Yaskawa INFORM job: X2_57-69(2)(90,180).JBI

/JOB
//NAME X2_57-69(2)(90,180)
//POS
///NPOS 364,364,364,19,0,0
///TOOL 0
///POSTYPE PULSE
///PULSE
C00000=-2000,-108350,-112464,0,80055,0
C00001=117728,-108350,-112464,34609,80055,28580
C00002=124329,53851,34766,36826,59228,24303
C00003=124742,48200,29458,35015,59253,25605
C00004=132091,87021,68515,19398,44781,35491
C00005=131964,91219,74916,20112,43130,35046
C00006=131964,92220,77875,20603,41902,34745
C00007=131925,92203,77341,20509,42211,34802
C00008=131397,96741,83157,21411,41178,34254
C00009=131925,92203,77341,20509,42211,34802
C00010=132378,78684,56627,18262,47592,36223
C00011=132682,70057,46287,17529,49367,36706
C00012=119143,48210,55676,30149,44593,-20608
C00013=119357,47156,53956,26116,42767,-17551
C00014=120340,57080,66927,26977,39866,-17985
C00015=120719,61633,72965,27509,38514,-18256
C00016=120718,63903,77470,28475,37088,-18806
C00017=120500,60851,73214,27972,38091,-18544
C00018=120914,65321,78494,28289,37111,-18678
C00019=120500,60851,73214,27972,38091,-18544
C00020=119122,46332,54187,26526,42331,-17820
C00021=118999,38480,45168,29507,46176,-20252
C00022=119368,-115903,-71302,26914,50601,-18610
C00023=64607,-7982,-59747,-18064,104585,18556
C00024=122352,27346,-5631,2134,105537,41861
C00025=121432,26579,-2459,2110,103216,41509
C00026=121064,26360,-1109,2102,102282,41368
C00027=120094,26356,-1113,2104,102307,41040
C00028=120094,26183,380,2095,101300,41022
C00029=120094,26356,-1113,2104,102307,41040
C00030=121064,26360,-1109,2102,102282,41368
C00031=121064,26166,399,2092,101255,41350
C00032=120526,26160,392,2094,101269,41168
C00033=121064,26166,399,2092,101255,41350
C00034=121064,26360,-1109,2102,102282,41368
C00035=121432,26579,-2459,2110,103216,41509
C00036=122352,27346,-5631,2134,105537,41861
C00037=122404,27316,-5660,2134,105538,41879
C00038=121484,26548,-2490,2110,103217,41527
C00039=121116,26328,-1140,2102,102284,41386
C00040=119990,26323,-1145,2104,102313,41004
C00041=119990,26151,349,2095,101305,40987
C00042=119990,26323,-1145,2104,102313,41004
C00043=121116,26328,-1140,2102,102284,41386
C00044=121116,26236,467,2092,101248,41368
C00045=120578,26229,460,2094,101262,41186
C00046=121116,26236,467,2092,101248,41368
C00047=121116,26328,-1140,2102,102284,41386
C00048=121484,26548,-2490,2110,103217,41527
C00049=122404,27316,-5660,2134,105538,41879
C00050=64607,-7982,-59747,-18064,104585,18556
C00051=43259,-142284,-94849,68481,67043,45987
C00052=75789,-57542,-35879,68380,64193,60275
C00053=79378,-55423,-31936,68889,61283,60160
C00054=80801,-54484,-30299,69115,60133,60112
C00055=80803,-53463,-27973,69597,59790,59668
C00056=80780,-53792,-28606,69479,59888,59772
C00057=82380,-55228,-29381,69587,58724,59873
C00058=80801,-53699,-28530,69478,59874,59776
C00059=81788,-51404,-27272,69234,59369,60118
C00060=80801,-53699,-28530,69478,59874,59776
C00061=79378,-54655,-30185,69233,61022,59829
C00062=75790,-56818,-34168,68680,63927,59955
C00063=84853,-69188,-42023,59966,34850,64425
C00064=87616,-64026,-36454,59770,32751,64733
C00065=88672,-61932,-34175,59731,31934,64834
C00066=88674,-60834,-31833,60968,31481,64183
C00067=88651,-60985,-32132,60826,31549,64256
C00068=90372,-59623,-31443,59618,30637,65026
C00069=88651,-60985,-32132,60826,31549,64256
C00070=87595,-63088,-34428,60823,32369,64172
C00071=84831,-68269,-40036,60922,34477,63902
C00072=34135,-92769,-74242,67244,95299,48930
C00073=35401,-42276,-48954,68810,98599,53574
C00074=65945,-1100,7259,69270,87048,42040
C00075=68239,35,11214,69501,84806,41537
C00076=69159,585,12885,69624,83908,41331
C00077=69161,1574,15470,69708,83504,40864
C00078=69221,1430,14991,69696,83546,40967
C00079=70472,2033,15498,69808,82706,41122
C00080=69221,1430,14991,69696,83546,40967
C00081=68301,843,13280,69560,84443,41175
C00082=66008,-382,9232,69294,86686,41685
C00083=65045,17742,23285,68512,88220,38243
C00084=67089,19246,27753,68708,86083,37667
C00085=67908,20664,31476,68858,84932,37105
C00086=67909,21636,33893,68917,84551,36681
C00087=67870,21286,33093,68893,84697,36810
C00088=69603,21321,33122,69077,83544,37032
C00089=67870,21286,33093,68893,84697,36810
C00090=67052,20507,31108,68763,85558,37056
C00091=65008,18839,26451,68515,87704,37647
C00092=35401,-42276,-48954,68810,98599,53574
C00093=34135,-92769,-74242,67244,95299,48930
C00094=40047,-44089,-55446,21687,109798,-38511
C00095=62225,-62197,-88507,27498,109393,-46828
C00096=110162,-85165,-68253,22495,93568,-66447
C00097=113189,-87083,-65902,22697,90484,-65921
C00098=114452,-87710,-64890,22792,89260,-65692
C00099=114517,-85766,-62478,22795,88793,-65757
C00100=114452,-87710,-64890,22792,89260,-65692
C00101=114560,-85938,-62764,22799,88863,-65728
C00102=116855,-86136,-62847,22980,88180,-65021
C00103=114560,-85938,-62764,22799,88863,-65728
C00104=116037,-86901,-63721,22918,88541,-65250
C00105=115908,-89550,-64185,22909,87583,-65481
C00106=116037,-86901,-63721,22918,88541,-65250
C00107=114760,-86329,-64757,22823,89756,-65485
C00108=111694,-84556,-67168,22619,92819,-66026
C00109=100686,-82782,-64085,34767,78413,-50947
C00110=101124,-84756,-62575,46086,58567,-32836
C00111=105363,-79670,-59021,44782,56711,-31479
C00112=106963,-77579,-57544,44243,56028,-30951
C00113=107094,-75757,-55111,44466,55555,-31127
C00114=106963,-77579,-57544,44243,56028,-30951
C00115=107061,-76131,-55605,44423,55653,-31093
C00116=109164,-76621,-55827,43839,54522,-30514
C00117=107061,-76131,-55605,44423,55653,-31093
C00118=152521,-89404,-55591,-46164,31260,15215
C00119=151593,-87290,-55392,-44387,31486,14209
C00120=152521,-89404,-55591,-46164,31260,15215
C00121=153310,-92374,-57074,-47433,31236,15946
C00122=155515,-99823,-60624,-50849,31303,17939
C00123=144863,-106519,-66042,-48559,45403,33907
C00124=128223,-91539,-64179,-39651,61078,44936
C00125=123361,-87629,-60570,-38638,58731,43541
C00126=121491,-85978,-59075,-38202,57849,42987
C00127=121484,-83973,-56613,-38386,57460,43144
C00128=121491,-85978,-59075,-38202,57849,42987
C00129=121461,-84428,-57196,-38332,57549,43096
C00130=119429,-85653,-57392,-38005,56255,42626
C00131=121461,-84428,-57196,-38332,57549,43096
C00132=119967,-84308,-57809,-37774,57245,42484
C00133=118856,-82106,-57411,-37133,57477,41844
C00134=119967,-84308,-57809,-37774,57245,42484
C00135=121794,-85994,-59329,-38223,58099,43033
C00136=126552,-90004,-63001,-39273,60372,44418
C00137=126573,-96663,-78450,-37396,65213,42514
C00138=131304,-91681,-76533,-26004,78425,57156
C00139=124056,-87914,-75121,-11214,89260,70181
C00140=122142,-89367,-72002,-11215,86376,69779
C00141=121349,-89811,-70686,-11221,85247,69607
C00142=121343,-87912,-68316,-11227,84773,69647
C00143=121349,-89811,-70686,-11221,85247,69607
C00144=121327,-88368,-69271,-11223,85117,69610
C00145=121333,-89533,-69503,-11227,84670,69652
C00146=121327,-88658,-70019,-11219,85423,69583
C00147=119585,-89190,-70235,-11210,85043,69016
C00148=122145,-87062,-69869,-11216,86251,69790
C00149=120261,-90277,-71864,-11211,85572,69201
C00150=122240,-88980,-75059,-11209,88432,69628
C00151=122263,-92131,-88871,-11297,95190,69025
C00152=118027,-102145,-112609,12133,81631,15728
C00153=114779,-111065,-98137,30741,51344,-26323
C00154=118307,-102289,-93656,28063,51644,-24513
C00155=119601,-98864,-91828,27075,51783,-23857
C00156=119613,-97097,-89588,27235,51358,-23975
C00157=119601,-98864,-91828,27075,51783,-23857
C00158=110485,-79839,-84525,36111,67748,-27732
C00159=112543,-80296,-84732,35339,66815,-27160
C00160=110485,-79839,-84525,36111,67748,-27732
C00161=133496,-108715,-92181,7385,37609,-14213
C00162=133101,-105069,-91479,7525,39076,-14289
C00163=133496,-108715,-92181,7385,37609,-14213
C00164=132876,-112861,-94058,8163,36703,-14650
C00165=131137,-123655,-98655,10535,34221,-15975
C00166=123443,-118355,-110381,19336,67280,-34215
C00167=114391,-92529,-101967,29874,101827,-55519
C00168=118393,-95739,-100418,29397,98177,-54940
C00169=120031,-96781,-99698,29226,96757,-54678
C00170=120038,-95275,-97552,29185,96274,-54799
C00171=120031,-96781,-99698,29226,96757,-54678
C00172=120084,-95528,-97941,29191,96355,-54761
C00173=122387,-95485,-97926,29054,95580,-54078
C00174=120084,-95528,-97941,29191,96355,-54761
C00175=120976,-97030,-99100,29136,95998,-54511
C00176=120991,-101427,-100201,29036,94603,-54858
C00177=120976,-97030,-99100,29136,95998,-54511
C00178=119331,-96066,-99851,29302,97402,-54781
C00179=115306,-93056,-101481,29762,101015,-55383
C00180=119500,-95286,-111088,6725,93490,-23573
C00181=126773,-109990,-105967,-32242,60764,29595
C00182=122699,-100871,-93398,-31267,56629,29081
C00183=121186,-97859,-91654,-30361,56488,28429
C00184=121181,-96122,-89420,-30519,56067,28559
C00185=121186,-97859,-91654,-30361,56488,28429
C00186=121151,-96393,-89780,-30476,56128,28526
C00187=118823,-96364,-89767,-29286,55307,27705
C00188=121151,-96393,-89780,-30476,56128,28526
C00189=120304,-96962,-90655,-29967,56039,28163
C00190=120309,-93163,-89734,-29527,57250,27795
C00191=120304,-96962,-90655,-29967,56039,28163
C00192=121790,-99973,-92408,-30869,56167,28809
C00193=125792,-107589,-96692,-33228,56592,30543
C00194=131625,-94984,-104332,-26399,91581,50246
C00195=126745,-145288,-119778,-15495,97214,71135
C00196=123697,-150191,-117695,-15760,92961,70600
C00197=122386,-151760,-116729,-15896,91357,70347
C00198=122362,-148095,-114205,-15905,91670,70298
C00199=122386,-151760,-116729,-15896,91357,70347
C00200=152021,-159898,-112636,-26025,88694,79156
C00201=148454,-161901,-113048,-26644,86894,78253
C00202=152021,-159898,-112636,-26025,88694,79156
C00203=97626,-122802,-108845,-7114,105595,63457
C00204=96843,-127398,-109672,-7190,103687,63292
C00205=97626,-122802,-108845,-7114,105595,63457
C00206=98540,-120520,-109456,-7005,107212,63690
C00207=100688,-114056,-110651,-6782,111424,64223
C00208=141928,-132033,-122827,-28072,87297,56565
C00209=127745,-107087,-104050,-36954,70100,33758
C00210=123019,-101123,-100201,-35200,68701,32195
C00211=121229,-98695,-98613,-34495,68204,31593
C00212=121224,-97088,-96437,-34605,67775,31733
C00213=121229,-98695,-98613,-34495,68204,31593
C00214=121227,-97196,-96702,-34583,67865,31704
C00215=118899,-97170,-96690,-33712,66948,31006
C00216=121227,-97196,-96702,-34583,67865,31704
C00217=120189,-96862,-97597,-34041,68055,31198
C00218=120197,-92600,-96484,-33733,69318,30794
C00219=120189,-96862,-97597,-34041,68055,31198
C00220=121940,-99293,-99200,-34743,68533,31788
C00221=126568,-105279,-103092,-36497,69877,33324
C00222=126928,-101255,-99744,-25325,80548,44815
C00223=122663,-98736,-96036,-24420,78380,43689
C00224=120996,-97606,-94499,-24052,77561,43237
C00225=120993,-95941,-92294,-24092,77100,43331
C00226=120996,-97606,-94499,-24052,77561,43237
C00227=121020,-96262,-92743,-24089,77210,43319
C00228=118702,-96225,-92727,-23520,76555,42587
C00229=121020,-96262,-92743,-24089,77210,43319
C00230=122674,-97386,-94282,-24452,78030,43766
C00231=126903,-99897,-97999,-25343,80198,44881
C00232=120621,-96600,-101484,-24088,62946,45857
C00233=120621,-96804,-99274,-24394,61605,46162
C00234=121065,-96725,-98290,-24739,61217,46434
C00235=120808,-96049,-104031,-23738,79088,41099
C00236=120748,-96229,-90224,-24572,71199,42719
C00237=112992,-105726,-101839,-14067,93209,37194
C00238=115215,-122388,-108196,-15088,94657,37910
C00239=120621,-96757,-99844,-19967,111704,37232
C00240=139470,-90927,-100236,-32127,92639,54211
C00241=120586,-139946,-100537,-59993,22470,77721
C00242=120585,-131753,-89573,-65663,21254,80445
C00243=120585,-129979,-87167,-67023,21013,81095
C00244=120562,-131266,-88538,-66553,21075,80878
C00245=122227,-132208,-89206,-62791,23886,78792
C00246=121243,-147626,-110329,-33756,48909,60234
C00247=120920,-140051,-100583,-34677,47022,60829
C00248=124359,-147547,-111068,-11567,101442,53176
C00249=120588,-147693,-110556,-9391,106075,51659
C00250=120588,-150839,-114378,-9432,106801,51602
C00251=120668,-127498,-127599,8027,92338,11843
C00252=106540,-131828,-115388,26739,62994,-22536
C00253=120606,-112501,-85686,37507,17849,-56930
C00254=120605,-109780,-80480,41231,16435,-58666
C00255=120605,-108994,-78986,42415,16045,-59215
C00256=120315,-109307,-78838,43536,15999,-59746
C00257=120588,-122985,-110649,24761,70026,-42850
C00258=120328,-120662,-104365,25254,67672,-43482
C00259=120364,-122737,-110073,20558,99126,-39146
C00260=120608,-123337,-111674,20610,99768,-38950
C00261=120609,-124066,-114983,20744,101328,-38677
C00262=120610,-124421,-123392,21260,106003,-37833
C00263=120649,-125888,-127056,5137,96316,-15534
C00264=120651,-130620,-101533,-26318,65901,27317
C00265=132080,-98652,-65915,-40871,60604,46715
C00266=126739,-94814,-62411,-39928,58019,45199
C00267=125167,-93744,-61263,-39656,57186,44775
C00268=114973,-73674,-63266,-21215,75827,54043
C00269=129996,-102072,-68542,-24583,69504,61007
C00270=129963,-88454,-64083,-24262,79764,67113
C00271=119249,-73873,-63371,-13635,90655,67540
C00272=119873,-76495,-66852,-13633,91534,67660
C00273=119888,-78331,-76038,-13747,96118,67156
C00274=119081,-108028,-88031,16388,61795,15984
C00275=117234,-100128,-64028,47858,30144,-31364
C00276=117223,-96877,-58390,50267,28944,-32603
C00277=120408,-90078,-55153,45893,28312,-30090
C00278=121323,-87057,-53987,43493,28946,-29243
C00279=115884,-56336,-58001,25875,73139,-43981
C00280=110450,-120996,-68796,34057,51702,-52465
C00281=115886,-81683,-60397,23196,86120,-63160
C00282=116435,-73198,-57641,22557,92556,-65246
C00283=113722,-71149,-59788,22419,95499,-65689
C00284=113460,-61701,-78205,24579,95746,-61766
C00285=45876,-101964,-103313,26325,110018,-55581
C00286=15431,-40197,-19183,56345,102197,5038
C00287=34862,-44642,-10243,68104,90731,26909
C00288=38272,-42530,-5806,68888,87904,26638
C00289=46229,766,28384,61909,108262,28635
C00290=46231,618,28261,61910,108260,28636
C00291=41809,-20527,11988,64520,102557,33043
C00292=37345,-41369,-1566,65704,98540,31804
C00293=38123,-41321,-1546,64762,100173,32421
C00294=38612,-39929,-4176,63239,100836,34262
C00295=36669,-38826,-14631,64435,105300,36937
C00296=35614,-75221,-31334,66701,43579,46020
C00297=-4350,-87290,-51239,65137,72622,41765
C00298=64440,-113176,-91621,27014,43904,67647
C00299=122842,55452,53671,34630,66319,-4477
C00300=122836,62423,70424,36514,60793,-6445
C00301=123914,74645,87958,37956,56708,-7549
C00302=125197,76616,91296,38180,55337,-7504
C00303=125636,70432,83250,33590,52050,-4701
C00304=125796,66906,78975,31139,50064,-1893
C00305=125404,66054,77985,29591,48689,-234
C00306=125098,65276,77131,27878,47332,1494
C00307=124827,64021,75593,26067,46325,3194
C00308=126696,59695,70609,19763,43762,8616
C00309=131143,56273,67245,5204,39677,20871
C00310=133431,54832,66811,-3343,37312,26727
C00311=136536,53744,67301,-15167,35496,34368
C00312=138731,52021,65734,-21083,35846,38135
C00313=139736,44763,55186,-20533,38686,37917
C00314=132675,46810,50748,6411,52596,1677
C00315=131127,80601,47453,25263,64319,31877
C00316=132807,97166,57058,12495,61470,40417
C00317=132437,103413,60649,12594,62499,40395
C00318=132694,105523,62562,12460,62371,40474
C00319=135614,121161,83227,11303,57371,41050
C00320=136368,126562,90481,11059,55609,41167
C00321=135950,123674,72731,10332,64945,41919
C00322=131127,80601,47453,25263,64319,31877
C00323=64440,-113176,-91621,27014,43904,67647
C00324=-4350,-87290,-51239,65137,72622,41765
C00325=52724,-99155,-43299,70564,49554,58260
C00326=58609,-95164,-38578,71970,45609,58601
C00327=62335,-94288,-36780,73026,43083,58718
C00328=62099,-93953,-36639,72913,43256,58740
C00329=60961,-88486,-31404,79687,39616,52248
C00330=56515,-82230,-27602,80423,44365,48776
C00331=50142,-68435,-18604,81559,53334,41178
C00332=51696,-72558,-17243,91450,48356,32919
C00333=47167,-82165,-29359,87907,51434,34351
C00334=62742,-127620,-60643,64448,25144,51124
C00335=120681,-113766,-68295,5608,40697,75829
C00336=102629,-70164,-59862,1874,75871,45222
C00337=101346,-35641,-42715,497,87745,38363
C00338=108372,-47074,-47716,-765,88535,35936
C00339=106813,-45162,-42766,-663,86458,35421
C00340=106148,-44305,-40721,-618,85635,35200
C00341=108217,-21947,-25956,-755,88052,35887
C00342=108724,-23055,-28269,-789,88913,36052
C00343=110078,-24539,-33116,-879,91147,36494
C00344=108372,-47074,-47716,-765,88535,35936
C00345=106813,-45162,-42766,-663,86458,35421
C00346=106197,-44302,-40640,-622,85587,35216
C00347=108187,-22349,-26070,-753,87917,35877
C00348=108724,-23055,-28269,-789,88913,36052
C00349=110078,-24539,-33116,-879,91147,36494
C00350=110090,-24487,-41377,-887,96257,36462
C00351=139155,108093,66847,-28518,79904,-60930
C00352=134264,102315,60055,-26951,79409,-62630
C00353=134200,103488,65613,-27168,76866,-62058
C00354=134676,107359,72292,-27534,75125,-61461
C00355=134682,108402,73653,-27571,74857,-61391
C00356=121037,104422,68475,-22889,71801,-65893
C00357=121135,105044,77589,-27533,52828,-61382
C00358=122558,77493,34057,-25010,64663,-63822
C00359=125010,77863,34506,-26345,65303,-63027
C00360=124245,5305,-48230,-24095,77496,-66005
C00361=134466,-50257,-37576,-52189,48931,-20490
C00362=81076,-72659,-48421,-23430,47332,-22731
C00363=-421,-73083,-90384,286,80877,488
BC00000=30026,523905,620826
BC00001=128747,520298,393743
BC00002=128747,400556,393743
BC00003=128747,406357,309655
BC00004=128747,400556,267992
BC00005=128747,400556,267992
BC00006=128747,400556,267992
BC00007=128747,400556,267992
BC00008=128747,400556,267992
BC00009=128747,400556,267992
BC00010=128747,400556,267992
BC00011=128747,400556,267992
BC00012=117613,412965,281863
BC00013=112293,418232,272920
BC00014=112293,418232,272920
BC00015=112293,418232,272920
BC00016=112293,418232,272920
BC00017=112293,418232,272920
BC00018=112293,418232,272920
BC00019=112293,418232,272920
BC00020=112293,418232,272920
BC00021=117955,415990,541185
BC00022=117955,517175,566904
BC00023=154514,517747,58960
BC00024=300288,515882,200400
BC00025=300288,515882,200400
BC00026=300288,515882,200400
BC00027=300288,515882,200400
BC00028=300288,515882,200400
BC00029=300288,515882,200400
BC00030=300288,515882,200400
BC00031=300288,515882,200400
BC00032=300288,515882,200400
BC00033=300288,515882,200400
BC00034=300288,515882,200400
BC00035=300288,515882,200400
BC00036=300288,515882,200400
BC00037=300597,468689,201286
BC00038=300597,468689,201286
BC00039=300597,468689,201286
BC00040=300597,468689,201286
BC00041=300597,468689,201286
BC00042=300597,468689,201286
BC00043=300597,468689,201286
BC00044=300597,468689,201286
BC00045=300597,468689,201286
BC00046=300597,468689,201286
BC00047=300597,468689,201286
BC00048=300597,468689,201286
BC00049=300597,468689,201286
BC00050=154514,517747,58960
BC00051=398158,497885,24767
BC00052=398158,523889,198574
BC00053=398158,523889,198574
BC00054=398158,523889,198574
BC00055=398158,523889,198574
BC00056=398158,523889,198574
BC00057=398158,523889,198574
BC00058=398158,523889,198574
BC00059=398158,523889,198574
BC00060=398158,523889,198574
BC00061=398158,523889,198574
BC00062=398158,523889,198574
BC00063=398158,523889,211671
BC00064=398158,523889,211671
BC00065=398158,523889,211671
BC00066=398158,523889,211671
BC00067=398158,523889,211671
BC00068=398158,523889,211671
BC00069=398158,523889,211671
BC00070=398158,523889,211671
BC00071=398158,523889,211671
BC00072=398158,488247,55914
BC00073=398158,488247,55914
BC00074=398158,523889,226332
BC00075=398158,523889,226332
BC00076=398158,523889,226332
BC00077=398158,523889,226332
BC00078=398158,523889,226332
BC00079=398158,523889,226332
BC00080=398158,523889,226332
BC00081=398158,523889,226332
BC00082=398158,523889,226332
BC00083=398158,523889,232778
BC00084=398158,523889,232778
BC00085=398158,523889,232778
BC00086=398158,523889,232778
BC00087=398158,523889,232778
BC00088=398158,523889,232778
BC00089=398158,523889,232778
BC00090=398158,523889,232778
BC00091=398158,523889,232778
BC00092=398158,488247,55914
BC00093=398158,488247,55914
BC00094=293957,522128,1025224
BC00095=329838,495468,1042664
BC00096=398158,462104,1075139
BC00097=398158,462104,1075139
BC00098=398158,462104,1075139
BC00099=398158,462104,1075139
BC00100=398158,462104,1075139
BC00101=398158,462104,1075139
BC00102=398158,462104,1075139
BC00103=398158,462104,1075139
BC00104=398158,462104,1075139
BC00105=398158,462104,1075139
BC00106=398158,462104,1075139
BC00107=398158,462104,1075139
BC00108=398158,462104,1075139
BC00109=396788,469265,1075139
BC00110=395417,476425,1075139
BC00111=395417,476425,1075139
BC00112=395417,476425,1075139
BC00113=395417,476425,1075139
BC00114=395417,476425,1075139
BC00115=395417,476425,1075139
BC00116=395417,476425,1075139
BC00117=395417,476425,1075139
BC00118=395417,476425,1075139
BC00119=395417,476425,1075139
BC00120=395417,476425,1075139
BC00121=395417,476425,1075139
BC00122=395417,476425,1075139
BC00123=386331,482370,1075139
BC00124=377245,488314,1075139
BC00125=377245,488314,1075139
BC00126=377245,488314,1075139
BC00127=377245,488314,1075139
BC00128=377245,488314,1075139
BC00129=377245,488314,1075139
BC00130=377245,488314,1075139
BC00131=377245,488314,1075139
BC00132=377245,488314,1075139
BC00133=377245,488314,1075139
BC00134=377245,488314,1075139
BC00135=377245,488314,1075139
BC00136=377245,488314,1075139
BC00137=377245,488314,1075139
BC00138=386461,479522,1075139
BC00139=397095,469378,1075139
BC00140=397095,469378,1075139
BC00141=397095,469378,1075139
BC00142=397095,469378,1075139
BC00143=397095,469378,1075139
BC00144=397095,469378,1075139
BC00145=397095,469378,1075139
BC00146=397095,469378,1075139
BC00147=397095,469378,1075139
BC00148=397095,469378,1075139
BC00149=397095,469378,1075139
BC00150=397095,469378,1075139
BC00151=397095,469378,1075139
BC00152=341534,401475,1075139
BC00153=299864,350547,1075139
BC00154=299864,350547,1075139
BC00155=299864,350547,1075139
BC00156=299864,350547,1075139
BC00157=299864,350547,1075139
BC00158=299864,350547,1075139
BC00159=299864,350547,1075139
BC00160=299864,350547,1075139
BC00161=299864,350547,1075139
BC00162=299864,350547,1075139
BC00163=299864,350547,1075139
BC00164=299864,350547,1075139
BC00165=299864,350547,1075139
BC00166=307766,330457,1075139
BC00167=316721,307688,1075139
BC00168=316721,307688,1075139
BC00169=316721,307688,1075139
BC00170=316721,307688,1075139
BC00171=316721,307688,1075139
BC00172=316721,307688,1075139
BC00173=316721,307688,1075139
BC00174=316721,307688,1075139
BC00175=316721,307688,1075139
BC00176=316721,307688,1075139
BC00177=316721,307688,1075139
BC00178=316721,307688,1075139
BC00179=316721,307688,1075139
BC00180=292119,323167,1075139
BC00181=249067,350254,1075139
BC00182=249067,350254,1075139
BC00183=249067,350254,1075139
BC00184=249067,350254,1075139
BC00185=249067,350254,1075139
BC00186=249067,350254,1075139
BC00187=249067,350254,1075139
BC00188=249067,350254,1075139
BC00189=249067,350254,1075139
BC00190=249067,350254,1075139
BC00191=249067,350254,1075139
BC00192=249067,350254,1075139
BC00193=249067,350254,1075139
BC00194=258766,329546,1075139
BC00195=268465,276709,1075139
BC00196=268465,276709,1075139
BC00197=268465,276709,1075139
BC00198=268465,276709,1075139
BC00199=268465,276709,1075139
BC00200=268465,276709,1075139
BC00201=268465,276709,1075139
BC00202=268465,276709,1075139
BC00203=268465,276709,1075139
BC00204=268465,276709,1075139
BC00205=268465,276709,1075139
BC00206=268465,276709,1075139
BC00207=268465,276709,1075139
BC00208=278919,312113,1075139
BC00209=286865,339020,1075139
BC00210=286865,339020,1075139
BC00211=286865,339020,1075139
BC00212=286865,339020,1075139
BC00213=286865,339020,1075139
BC00214=286865,339020,1075139
BC00215=286865,339020,1075139
BC00216=286865,339020,1075139
BC00217=286865,339020,1075139
BC00218=286865,339020,1075139
BC00219=286865,339020,1075139
BC00220=286865,339020,1075139
BC00221=286865,339020,1075139
BC00222=299147,390471,1075139
BC00223=299147,390471,1075139
BC00224=299147,390471,1075139
BC00225=299147,390471,1075139
BC00226=299147,390471,1075139
BC00227=299147,390471,1075139
BC00228=299147,390471,1075139
BC00229=299147,390471,1075139
BC00230=299147,390471,1075139
BC00231=299147,390471,1075139
BC00232=297684,353023,1075139
BC00233=303127,349350,1075139
BC00234=305304,347880,1075139
BC00235=302218,329336,1075139
BC00236=302023,399288,1075139
BC00237=308205,358158,1075139
BC00238=309127,337938,1075139
BC00239=304033,336581,1075139
BC00240=283556,352227,1075139
BC00241=252387,344292,1075139
BC00242=252408,344289,1075139
BC00243=257433,339351,1075139
BC00244=259443,337375,1075139
BC00245=258584,334701,1075139
BC00246=250395,309217,1075139
BC00247=250348,347410,1075139
BC00248=276218,261338,1075139
BC00249=277667,249884,1075139
BC00250=273915,245784,1075139
BC00251=280029,300408,1075139
BC00252=284276,326768,1075139
BC00253=290087,362839,1075139
BC00254=290097,362838,1075139
BC00255=285795,356754,1075139
BC00256=284075,354321,1075139
BC00257=306175,301342,1075139
BC00258=306092,331294,1075139
BC00259=300548,281510,1075139
BC00260=302655,281119,1075139
BC00261=307955,280438,1075139
BC00262=307934,280441,1075139
BC00263=326059,338602,1075139
BC00264=360985,450671,1075139
BC00265=387153,477098,1075139
BC00266=387153,477098,1075139
BC00267=387153,477098,1075139
BC00268=387153,477098,1075139
BC00269=387153,477098,1075139
BC00270=387153,477098,1075139
BC00271=387153,477098,1075139
BC00272=387153,477098,1075139
BC00273=387153,477098,1075139
BC00274=393633,477999,1075139
BC00275=397752,474419,1075139
BC00276=397752,474419,1075139
BC00277=397752,474419,1075139
BC00278=397752,474419,1075139
BC00279=397752,474419,1075139
BC00280=397752,474419,1075139
BC00281=397752,474419,1075139
BC00282=397752,474419,1075139
BC00283=397752,474419,1075139
BC00284=398158,494487,1075139
BC00285=369887,500848,936014
BC00286=391319,465889,463853
BC00287=398158,441448,291370
BC00288=398158,441448,291370
BC00289=398158,441448,291370
BC00290=398158,441448,291370
BC00291=398158,441448,291370
BC00292=398158,441448,291370
BC00293=398158,441448,291370
BC00294=398158,441448,291370
BC00295=398158,441448,291370
BC00296=398158,450952,312705
BC00297=328719,450952,312705
BC00298=38883,521356,566128
BC00299=131006,403465,300248
BC00300=131006,403465,300248
BC00301=131006,403465,300248
BC00302=131006,403465,300248
BC00303=131006,403465,300248
BC00304=131006,403465,300248
BC00305=131006,403465,300248
BC00306=131006,403465,300248
BC00307=131006,403465,300248
BC00308=131006,403465,300248
BC00309=131006,403465,300248
BC00310=131006,403465,300248
BC00311=131006,403465,300248
BC00312=131006,403465,300248
BC00313=131006,403465,300248
BC00314=135578,398427,312903
BC00315=142497,416817,255630
BC00316=135849,405323,149549
BC00317=135849,405323,97845
BC00318=135849,405323,85978
BC00319=135849,405323,85978
BC00320=135849,405323,85978
BC00321=135849,405323,4459
BC00322=142497,416817,255630
BC00323=38883,521356,566128
BC00324=328719,450952,312705
BC00325=368722,473501,285123
BC00326=368722,473501,285123
BC00327=368722,473501,285123
BC00328=368722,473501,285123
BC00329=368722,473501,285123
BC00330=368722,473501,285123
BC00331=368722,473501,285123
BC00332=368722,473501,285123
BC00333=368722,473501,285123
BC00334=369539,481975,264435
BC00335=300471,495640,304855
BC00336=255606,449497,293914
BC00337=261418,454966,291041
BC00338=265736,459028,288906
BC00339=265736,459028,288906
BC00340=265736,459028,288906
BC00341=265736,459028,288906
BC00342=265736,459028,288906
BC00343=265736,459028,288906
BC00344=265891,411979,289791
BC00345=265891,411979,289791
BC00346=265891,411979,289791
BC00347=265891,411979,289791
BC00348=265891,411979,289791
BC00349=265891,411979,289791
BC00350=265891,411979,289791
BC00351=338854,523889,48764
BC00352=338874,523889,17
BC00353=340241,523889,17
BC00354=340788,523889,17
BC00355=340803,521511,17
BC00356=286951,445210,17
BC00357=286951,445210,17
BC00358=286951,464032,17
BC00359=286951,556384,17
BC00360=286951,556384,17
BC00361=303352,548024,298275
BC00362=255922,546396,377431
BC00363=146427,523905,652589
EC00000=-798156,-1296783
EC00001=-798156,-1296783
EC00002=-798156,-1296783
EC00003=-798156,-1296783
EC00004=-798156,-1296783
EC00005=-798156,-1296783
EC00006=-798156,-1296783
EC00007=-798156,-1296783
EC00008=-798156,-1296783
EC00009=-798156,-1296783
EC00010=-798156,-1296783
EC00011=-798156,-1296783
EC00012=-798156,-1296783
EC00013=-798156,-1296783
EC00014=-798156,-1296783
EC00015=-798156,-1296783
EC00016=-798156,-1296783
EC00017=-798156,-1296783
EC00018=-798156,-1296783
EC00019=-798156,-1296783
EC00020=-798156,-1296783
EC00021=-798156,-1296783
EC00022=-798156,-1296783
EC00023=-798156,-1296783
EC00024=-798156,-1296783
EC00025=-798156,-1296783
EC00026=-798156,-1296783
EC00027=-798156,-1296783
EC00028=-798156,-1296783
EC00029=-798156,-1296783
EC00030=-798156,-1296783
EC00031=-798156,-1296783
EC00032=-798156,-1296783
EC00033=-798156,-1296783
EC00034=-798156,-1296783
EC00035=-798156,-1296783
EC00036=-798156,-1296783
EC00037=-798156,-1296783
EC00038=-798156,-1296783
EC00039=-798156,-1296783
EC00040=-798156,-1296783
EC00041=-798156,-1296783
EC00042=-798156,-1296783
EC00043=-798156,-1296783
EC00044=-798156,-1296783
EC00045=-798156,-1296783
EC00046=-798156,-1296783
EC00047=-798156,-1296783
EC00048=-798156,-1296783
EC00049=-798156,-1296783
EC00050=-798156,-1296783
EC00051=-798156,-1296783
EC00052=-798156,-1296783
EC00053=-798156,-1296783
EC00054=-798156,-1296783
EC00055=-798156,-1296783
EC00056=-798156,-1296783
EC00057=-798156,-1296783
EC00058=-798156,-1296783
EC00059=-798156,-1296783
EC00060=-798156,-1296783
EC00061=-798156,-1296783
EC00062=-798156,-1296783
EC00063=-798156,-1296783
EC00064=-798156,-1296783
EC00065=-798156,-1296783
EC00066=-798156,-1296783
EC00067=-798156,-1296783
EC00068=-798156,-1296783
EC00069=-798156,-1296783
EC00070=-798156,-1296783
EC00071=-798156,-1296783
EC00072=-798156,-1296783
EC00073=-798156,-1296783
EC00074=-798156,-1296783
EC00075=-798156,-1296783
EC00076=-798156,-1296783
EC00077=-798156,-1296783
EC00078=-798156,-1296783
EC00079=-798156,-1296783
EC00080=-798156,-1296783
EC00081=-798156,-1296783
EC00082=-798156,-1296783
EC00083=-798156,-1296783
EC00084=-798156,-1296783
EC00085=-798156,-1296783
EC00086=-798156,-1296783
EC00087=-798156,-1296783
EC00088=-798156,-1296783
EC00089=-798156,-1296783
EC00090=-798156,-1296783
EC00091=-798156,-1296783
EC00092=-798156,-1296783
EC00093=-798156,-1296783
EC00094=-912440,-1296783
EC00095=-934482,-1296783
EC00096=-975524,-1296783
EC00097=-975524,-1296783
EC00098=-975524,-1296783
EC00099=-975524,-1296783
EC00100=-975524,-1296783
EC00101=-975524,-1296783
EC00102=-975524,-1296783
EC00103=-975524,-1296783
EC00104=-975524,-1296783
EC00105=-975524,-1296783
EC00106=-975524,-1296783
EC00107=-975524,-1296783
EC00108=-975524,-1296783
EC00109=-975524,-1296783
EC00110=-975524,-1296783
EC00111=-975524,-1296783
EC00112=-975524,-1296783
EC00113=-975524,-1296783
EC00114=-975524,-1296783
EC00115=-975524,-1296783
EC00116=-975524,-1296783
EC00117=-975524,-1296783
EC00118=-975524,-1296783
EC00119=-975524,-1296783
EC00120=-975524,-1296783
EC00121=-975524,-1296783
EC00122=-975524,-1296783
EC00123=-975524,-1296783
EC00124=-975524,-1296783
EC00125=-975524,-1296783
EC00126=-975524,-1296783
EC00127=-975524,-1296783
EC00128=-975524,-1296783
EC00129=-975524,-1296783
EC00130=-975524,-1296783
EC00131=-975524,-1296783
EC00132=-975524,-1296783
EC00133=-975524,-1296783
EC00134=-975524,-1296783
EC00135=-975524,-1296783
EC00136=-975524,-1296783
EC00137=-975524,-1296783
EC00138=-975524,-1296783
EC00139=-975524,-1296783
EC00140=-975524,-1296783
EC00141=-975524,-1296783
EC00142=-975524,-1296783
EC00143=-975524,-1296783
EC00144=-975524,-1296783
EC00145=-975524,-1296783
EC00146=-975524,-1296783
EC00147=-975524,-1296783
EC00148=-975524,-1296783
EC00149=-975524,-1296783
EC00150=-975524,-1296783
EC00151=-975524,-1296783
EC00152=-975524,-1296783
EC00153=-975524,-1296783
EC00154=-975524,-1296783
EC00155=-975524,-1296783
EC00156=-975524,-1296783
EC00157=-975524,-1296783
EC00158=-975524,-1296783
EC00159=-975524,-1296783
EC00160=-975524,-1296783
EC00161=-975524,-1296783
EC00162=-975524,-1296783
EC00163=-975524,-1296783
EC00164=-975524,-1296783
EC00165=-975524,-1296783
EC00166=-975524,-1296783
EC00167=-975524,-1296783
EC00168=-975524,-1296783
EC00169=-975524,-1296783
EC00170=-975524,-1296783
EC00171=-975524,-1296783
EC00172=-975524,-1296783
EC00173=-975524,-1296783
EC00174=-975524,-1296783
EC00175=-975524,-1296783
EC00176=-975524,-1296783
EC00177=-975524,-1296783
EC00178=-975524,-1296783
EC00179=-975524,-1296783
EC00180=-975524,-1296783
EC00181=-975524,-1296783
EC00182=-975524,-1296783
EC00183=-975524,-1296783
EC00184=-975524,-1296783
EC00185=-975524,-1296783
EC00186=-975524,-1296783
EC00187=-975524,-1296783
EC00188=-975524,-1296783
EC00189=-975524,-1296783
EC00190=-975524,-1296783
EC00191=-975524,-1296783
EC00192=-975524,-1296783
EC00193=-975524,-1296783
EC00194=-975524,-1296783
EC00195=-975524,-1296783
EC00196=-975524,-1296783
EC00197=-975524,-1296783
EC00198=-975524,-1296783
EC00199=-975524,-1296783
EC00200=-975524,-1296783
EC00201=-975524,-1296783
EC00202=-975524,-1296783
EC00203=-975524,-1296783
EC00204=-975524,-1296783
EC00205=-975524,-1296783
EC00206=-975524,-1296783
EC00207=-975524,-1296783
EC00208=-975524,-1296783
EC00209=-975524,-1296783
EC00210=-975524,-1296783
EC00211=-975524,-1296783
EC00212=-975524,-1296783
EC00213=-975524,-1296783
EC00214=-975524,-1296783
EC00215=-975524,-1296783
EC00216=-975524,-1296783
EC00217=-975524,-1296783
EC00218=-975524,-1296783
EC00219=-975524,-1296783
EC00220=-975524,-1296783
EC00221=-975524,-1296783
EC00222=-975524,-1296783
EC00223=-975524,-1296783
EC00224=-975524,-1296783
EC00225=-975524,-1296783
EC00226=-975524,-1296783
EC00227=-975524,-1296783
EC00228=-975524,-1296783
EC00229=-975524,-1296783
EC00230=-975524,-1296783
EC00231=-975524,-1296783
EC00232=-975524,-1296783
EC00233=-975524,-1296783
EC00234=-975524,-1296783
EC00235=-975524,-1296783
EC00236=-975524,-1296783
EC00237=-975524,-1296783
EC00238=-975524,-1296783
EC00239=-975524,-1296783
EC00240=-975524,-1296783
EC00241=-975524,-1296783
EC00242=-975524,-1296783
EC00243=-975524,-1296783
EC00244=-975522,-1296782
EC00245=-975524,-1296783
EC00246=-975524,-1296783
EC00247=-975524,-1296783
EC00248=-975524,-1296783
EC00249=-975524,-1296783
EC00250=-975524,-1296783
EC00251=-975524,-1296783
EC00252=-975524,-1296783
EC00253=-975524,-1296783
EC00254=-975524,-1296783
EC00255=-975524,-1296783
EC00256=-975524,-1296783
EC00257=-975524,-1296783
EC00258=-975524,-1296783
EC00259=-975524,-1296783
EC00260=-975524,-1296783
EC00261=-975524,-1296783
EC00262=-975524,-1296783
EC00263=-975524,-1296783
EC00264=-975524,-1296783
EC00265=-975524,-1296783
EC00266=-975524,-1296783
EC00267=-975524,-1296783
EC00268=-975524,-1296783
EC00269=-975524,-1296783
EC00270=-975523,-1296783
EC00271=-975524,-1296783
EC00272=-975524,-1296783
EC00273=-975524,-1296783
EC00274=-975524,-1296783
EC00275=-975524,-1296783
EC00276=-975524,-1296783
EC00277=-975524,-1296783
EC00278=-975524,-1296783
EC00279=-975524,-1296783
EC00280=-975524,-1296783
EC00281=-975524,-1296783
EC00282=-975524,-1296783
EC00283=-975524,-1296783
EC00284=-975524,-1296783
EC00285=-943270,-1296783
EC00286=-833264,-1296783
EC00287=-798156,-1296783
EC00288=-798156,-1296783
EC00289=-798156,-1296783
EC00290=-798156,-1296783
EC00291=-798156,-1296783
EC00292=-798156,-1296783
EC00293=-798156,-1296783
EC00294=-798156,-1296783
EC00295=-798156,-1296783
EC00296=-798156,-1296783
EC00297=-798156,-1296783
EC00298=-798156,-1296783
EC00299=-798156,-1296783
EC00300=-798156,-1296783
EC00301=-798156,-1296783
EC00302=-798156,-1296783
EC00303=-798156,-1296783
EC00304=-798156,-1296783
EC00305=-798156,-1296783
EC00306=-798156,-1296783
EC00307=-798156,-1296783
EC00308=-798156,-1296783
EC00309=-798156,-1296783
EC00310=-798156,-1296783
EC00311=-798156,-1296783
EC00312=-798156,-1296783
EC00313=-798156,-1296783
EC00314=-798156,-1296783
EC00315=-798156,-1296783
EC00316=-798156,-1296783
EC00317=-798156,-1296783
EC00318=-798156,-1296783
EC00319=-798156,-1296783
EC00320=-798156,-1296783
EC00321=-798156,-1296783
EC00322=-798156,-1296783
EC00323=-798156,-1296783
EC00324=-798156,-1296783
EC00325=-798156,-1296783
EC00326=-798156,-1296783
EC00327=-798156,-1296783
EC00328=-798156,-1296783
EC00329=-798156,-1296783
EC00330=-798156,-1296783
EC00331=-798156,-1296783
EC00332=-798156,-1296783
EC00333=-798156,-1296783
EC00334=-798156,-1296783
EC00335=-798156,-1296783
EC00336=-798156,-1296783
EC00337=-798156,-1296783
EC00338=-798156,-1296783
EC00339=-798156,-1296783
EC00340=-798156,-1296783
EC00341=-798156,-1296783
EC00342=-798156,-1296783
EC00343=-798156,-1296783
EC00344=-798156,-1296783
EC00345=-798156,-1296783
EC00346=-798156,-1296783
EC00347=-798156,-1296783
EC00348=-798156,-1296783
EC00349=-798156,-1296783
EC00350=-798156,-1296783
EC00351=-798156,-1296783
EC00352=-798156,-1296783
EC00353=-798156,-1296783
EC00354=-798156,-1296783
EC00355=-798156,-1296783
EC00356=-798156,-1296783
EC00357=-798156,-1296783
EC00358=-798156,-1296783
EC00359=-798156,-1296783
EC00360=-798156,-1296783
EC00361=-798156,-1296783
EC00362=-798156,-1296783
EC00363=-798156,-1296783
///POSTYPE BASE
///RECTAN
///RCONF 0,0,0,0,1,0,0,0,0,0,0,0,0,0,0,0,0,0,0,0,0,0,0,0
P00006=2.006,1.622,-0.565,0.0000,0.0000,0.0000
///RCONF 0,0,0,0,0,0,0,0,0,0,0,0,0,0,0,0,0,0,0,0,0,0,0,0
P00020=-8.957,15.102,6.369,0.0000,0.0000,0.0000
///RCONF 0,0,0,0,1,0,0,0,0,0,0,0,0,0,0,0,0,0,0,0,0,0,0,0
P00022=2.006,1.622,-0.565,0.0000,0.0000,0.0000
///RCONF 0,0,0,0,0,0,0,0,0,0,0,0,0,0,0,0,0,0,0,0,0,0,0,0
P00023=-2.957,-4.083,2.762,0.0000,0.0000,0.0000
P00024=-1.466,-0.226,-0.419,0.0000,0.0000,0.0000
P00025=3.643,0.007,-2.585,0.0000,0.0000,0.0000
P00026=2.644,0.055,-2.583,0.0000,0.0000,0.0000
P00031=-0.170,0.039,-0.647,0.0000,0.0000,0.0000
P00032=-0.423,0.157,3.222,0.0000,0.0000,0.0000
P00033=0.854,-1.099,3.047,0.0000,0.0000,0.0000
///RCONF 0,0,0,0,1,0,0,0,0,0,0,0,0,0,0,0,0,0,0,0,0,0,0,0
P00034=-8.151,9.743,-4.393,0.0000,0.0000,0.0000
///RCONF 0,0,0,0,0,0,0,0,0,0,0,0,0,0,0,0,0,0,0,0,0,0,0,0
P00035=0.390,-0.027,1.040,0.0000,0.0000,0.0000
P00036=-2.434,0.084,0.197,0.0000,0.0000,0.0000
P00037=-1.075,5.090,-3.949,0.0000,0.0000,0.0000
P00038=0.174,-1.527,-10.860,0.0000,0.0000,0.0000
P00039=-0.109,1.838,-0.266,0.0000,0.0000,0.0000
P00040=2.716,-0.016,3.014,0.0000,0.0000,0.0000
P00041=-0.109,0.014,0.966,0.0000,0.0000,0.0000
P00042=-0.220,0.371,-0.613,0.0000,0.0000,0.0000
//INST
///DATE 2024/12/11 12:36
///ATTR SC,RW
///GROUP1 RB1,BS1
///GROUP2 ST1
NOP
'X2_57-69(2)(90,180)
'Down
MOVJ C00000 BC00000 VJ=100.00  +MOVJ EC00000 VJ=100.00
MOVJ C00001 BC00001 VJ=100.00  +MOVJ EC00001 VJ=100.00
MOVJ C00002 BC00002 VJ=100.00  +MOVJ EC00002 VJ=100.00
'Path S4549
SFTOF3D
MOVJ C00003 BC00003 VJ=100.00  +MOVJ EC00003 VJ=100.00
MOVL C00004 BC00004 V=800.0  +MOVJ EC00004 VJ=100.00
SMOVL C00005 BC00005 V=166.7  +MOVJ EC00005
SREFP 3 C00006 BC00006  +REFP EC00006
CALL JOB:SEARCH-R1-S13D
SET P020 P006
SFTON3D P020
SMOVL C00007 BC00007 V=166.7  +MOVJ EC00007
SREFP 3 C00008 BC00008  +REFP EC00008
CALL JOB:SEARCH-R1-S13D
SET P020 P006
SFTON3D P020
SMOVL C00009 BC00009 V=166.7  +MOVJ EC00009
MOVL C00010 BC00010 V=1000.0  +MOVJ EC00010 VJ=100.00
'EndPath S4549
'Path S3846
SFTOF3D
MOVJ C00011 BC00011 VJ=100.00  +MOVJ EC00011 VJ=100.00
MOVJ C00012 BC00012 VJ=100.00  +MOVJ EC00012 VJ=100.00
'EndPath S3846
'Path S4550
SFTOF3D
MOVJ C00013 BC00013 VJ=100.00  +MOVJ EC00013 VJ=100.00
MOVL C00014 BC00014 V=800.0  +MOVJ EC00014 VJ=100.00
SMOVL C00015 BC00015 V=166.7  +MOVJ EC00015
SREFP 3 C00016 BC00016  +REFP EC00016
CALL JOB:SEARCH-R1-S13D
SET P022 P006
SFTON3D P022
SMOVL C00017 BC00017 V=166.7  +MOVJ EC00017
SREFP 3 C00018 BC00018  +REFP EC00018
CALL JOB:SEARCH-R1-S13D
SET P022 P006
SFTON3D P022
SMOVL C00019 BC00019 V=166.7  +MOVJ EC00019
MOVL C00020 BC00020 V=1000.0  +MOVJ EC00020 VJ=100.00
'EndPath S4550
MOVJ C00021 BC00021 VJ=100.00  +MOVJ EC00021 VJ=100.00
MOVJ C00022 BC00022 VJ=100.00  +MOVJ EC00022 VJ=100.00
MOVJ C00023 BC00023 VJ=100.00  +MOVJ EC00023 VJ=100.00
'Path S4663
SFTOF3D
COMM PAUSE
COMM MOVJ C00024 BC00024 VJ=100.00  +MOVJ EC00024 VJ=100.00
COMM MOVL C00025 BC00025 V=800.0  +MOVJ EC00025 VJ=100.00
COMM SMOVL C00026 BC00026 V=166.7  +MOVJ EC00026
COMM SMOVL C00027 BC00027 V=166.7  +MOVJ EC00027
COMM SREFP 3 C00028 BC00028  +REFP EC00028
COMM CALL JOB:SEARCH-R1-S13D
COMM SET P041 P006
COMM SFTON3D P041
COMM SMOVL C00029 BC00029 V=166.7  +MOVJ EC00029
COMM SMOVL C00030 BC00030 V=166.7  +MOVJ EC00030
COMM SMOVL C00031 BC00031 V=166.7  +MOVJ EC00031
COMM SREFP 3 C00032 BC00032  +REFP EC00032
COMM CALL JOB:SEARCH-R1-S13D
COMM SET P041 P006
COMM SFTON3D P041
COMM SMOVL C00033 BC00033 V=166.7  +MOVJ EC00033
COMM SMOVL C00034 BC00034 V=166.7  +MOVJ EC00034
COMM MOVL C00035 BC00035 V=800.0  +MOVJ EC00035 VJ=100.00
COMM MOVL C00036 BC00036 V=1000.0  +MOVJ EC00036 VJ=100.00
COMM 'EndPath S4663
COMM 'Path S4664
COMM SFTOF3D
COMM MOVJ C00037 BC00037 VJ=100.00  +MOVJ EC00037 VJ=100.00
COMM MOVL C00038 BC00038 V=800.0  +MOVJ EC00038 VJ=100.00
COMM SMOVL C00039 BC00039 V=166.7  +MOVJ EC00039
COMM SMOVL C00040 BC00040 V=166.7  +MOVJ EC00040
COMM SREFP 3 C00041 BC00041  +REFP EC00041
COMM CALL JOB:SEARCH-R1-S13D
COMM SET P042 P006
COMM SFTON3D P042
COMM SMOVL C00042 BC00042 V=166.7  +MOVJ EC00042
COMM SMOVL C00043 BC00043 V=166.7  +MOVJ EC00043
COMM SMOVL C00044 BC00044 V=166.7  +MOVJ EC00044
COMM SREFP 3 C00045 BC00045  +REFP EC00045
COMM CALL JOB:SEARCH-R1-S13D
COMM SET P042 P006
COMM SFTON3D P042
COMM SMOVL C00046 BC00046 V=166.7  +MOVJ EC00046
COMM SMOVL C00047 BC00047 V=166.7  +MOVJ EC00047
COMM MOVL C00048 BC00048 V=800.0  +MOVJ EC00048 VJ=100.00
COMM MOVL C00049 BC00049 V=1000.0  +MOVJ EC00049 VJ=100.00
COMM 'EndPath S4664
MOVJ C00050 BC00050 VJ=100.00  +MOVJ EC00050 VJ=100.00
MOVJ C00051 BC00051 VJ=100.00  +MOVJ EC00051 VJ=100.00
'Path S3853
SFTOF3D
MOVJ C00052 BC00052 VJ=100.00  +MOVJ EC00052 VJ=100.00
MOVL C00053 BC00053 V=800.0  +MOVJ EC00053 VJ=100.00
SMOVL C00054 BC00054 V=166.7  +MOVJ EC00054
SREFP 3 C00055 BC00055  +REFP EC00055
CALL JOB:SEARCH-R1-S13D
SET P023 P006
SFTON3D P023
SMOVL C00056 BC00056 V=166.7  +MOVJ EC00056
SREFP 3 C00057 BC00057  +REFP EC00057
CALL JOB:SEARCH-R1-S13D
SET P023 P006
SFTON3D P023
SMOVL C00058 BC00058 V=166.7  +MOVJ EC00058
SREFP 3 C00059 BC00059  +REFP EC00059
CALL JOB:SEARCH-R1-S13D
SET P023 P006
SFTON3D P023
SMOVL C00060 BC00060 V=166.7  +MOVJ EC00060
MOVL C00061 BC00061 V=800.0  +MOVJ EC00061 VJ=100.00
MOVL C00062 BC00062 V=1000.0  +MOVJ EC00062 VJ=100.00
'EndPath S3853
'Path S4665
SFTOF3D
MOVJ C00063 BC00063 VJ=100.00  +MOVJ EC00063 VJ=100.00
MOVL C00064 BC00064 V=800.0  +MOVJ EC00064 VJ=100.00
SMOVL C00065 BC00065 V=166.7  +MOVJ EC00065
SREFP 3 C00066 BC00066  +REFP EC00066
CALL JOB:SEARCH-R1-S13D
SET P024 P006
SFTON3D P024
SMOVL C00067 BC00067 V=166.7  +MOVJ EC00067
SREFP 3 C00068 BC00068  +REFP EC00068
CALL JOB:SEARCH-R1-S13D
SET P024 P006
SFTON3D P024
SMOVL C00069 BC00069 V=166.7  +MOVJ EC00069
MOVL C00070 BC00070 V=800.0  +MOVJ EC00070 VJ=100.00
MOVL C00071 BC00071 V=1000.0  +MOVJ EC00071 VJ=100.00
'EndPath S4665
MOVJ C00072 BC00072 VJ=100.00  +MOVJ EC00072 VJ=100.00
MOVJ C00073 BC00073 VJ=100.00  +MOVJ EC00073 VJ=100.00
'Path S3854
SFTOF3D
MOVJ C00074 BC00074 VJ=100.00  +MOVJ EC00074 VJ=100.00
MOVL C00075 BC00075 V=800.0  +MOVJ EC00075 VJ=100.00
SMOVL C00076 BC00076 V=166.7  +MOVJ EC00076
SREFP 3 C00077 BC00077  +REFP EC00077
CALL JOB:SEARCH-R1-S13D
SET P025 P006
SFTON3D P025
SMOVL C00078 BC00078 V=166.7  +MOVJ EC00078
SREFP 3 C00079 BC00079  +REFP EC00079
CALL JOB:SEARCH-R1-S13D
SET P025 P006
SFTON3D P025
SMOVL C00080 BC00080 V=166.7  +MOVJ EC00080
MOVL C00081 BC00081 V=800.0  +MOVJ EC00081 VJ=100.00
MOVL C00082 BC00082 V=1000.0  +MOVJ EC00082 VJ=100.00
'EndPath S3854
'Path S3855
SFTOF3D
MOVJ C00083 BC00083 VJ=100.00  +MOVJ EC00083 VJ=100.00
MOVL C00084 BC00084 V=800.0  +MOVJ EC00084 VJ=100.00
SMOVL C00085 BC00085 V=166.7  +MOVJ EC00085
SREFP 3 C00086 BC00086  +REFP EC00086
CALL JOB:SEARCH-R1-S13D
SET P026 P006
SFTON3D P026
SMOVL C00087 BC00087 V=166.7  +MOVJ EC00087
SREFP 3 C00088 BC00088  +REFP EC00088
CALL JOB:SEARCH-R1-S13D
SET P026 P006
SFTON3D P026
SMOVL C00089 BC00089 V=166.7  +MOVJ EC00089
MOVL C00090 BC00090 V=800.0  +MOVJ EC00090 VJ=100.00
MOVL C00091 BC00091 V=1000.0  +MOVJ EC00091 VJ=100.00
'EndPath S3855
MOVJ C00092 BC00092 VJ=100.00  +MOVJ EC00092 VJ=100.00
MOVJ C00093 BC00093 VJ=100.00  +MOVJ EC00093 VJ=100.00
'Up
MOVJ C00094 BC00094 VJ=100.00  +MOVJ EC00094 VJ=100.00
MOVJ C00095 BC00095 VJ=100.00  +MOVJ EC00095 VJ=100.00
'Path S3856
SFTOF3D
MOVJ C00096 BC00096 VJ=100.00  +MOVJ EC00096 VJ=100.00
MOVL C00097 BC00097 V=800.0  +MOVJ EC00097 VJ=100.00
SMOVL C00098 BC00098 V=166.7  +MOVJ EC00098
SREFP 3 C00099 BC00099  +REFP EC00099
CALL JOB:SEARCH-R1-S13D
SET P031 P006
SFTON3D P031
SMOVL C00100 BC00100 V=166.7  +MOVJ EC00100
SMOVL C00101 BC00101 V=166.7  +MOVJ EC00101
SREFP 3 C00102 BC00102  +REFP EC00102
CALL JOB:SEARCH-R1-S13D
SET P031 P006
SFTON3D P031
SMOVL C00103 BC00103 V=166.7  +MOVJ EC00103
SMOVL C00104 BC00104 V=166.7  +MOVJ EC00104
SREFP 3 C00105 BC00105  +REFP EC00105
CALL JOB:SEARCH-R1-S13D
SET P031 P006
SFTON3D P031
SMOVL C00106 BC00106 V=166.7  +MOVJ EC00106
MOVL C00107 BC00107 V=800.0  +MOVJ EC00107 VJ=100.00
MOVL C00108 BC00108 V=1000.0  +MOVJ EC00108 VJ=100.00
'EndPath S3856
MOVJ C00109 BC00109 VJ=100.00  +MOVJ EC00109 VJ=100.00
'Path S4666
SFTOF3D
MOVJ C00110 BC00110 VJ=100.00  +MOVJ EC00110 VJ=100.00
MOVL C00111 BC00111 V=800.0  +MOVJ EC00111 VJ=100.00
SMOVL C00112 BC00112 V=166.7  +MOVJ EC00112
SREFP 3 C00113 BC00113  +REFP EC00113
CALL JOB:SEARCH-R1-S13D
SET P032 P006
SFTON3D P032
SMOVL C00114 BC00114 V=166.7  +MOVJ EC00114
SMOVL C00115 BC00115 V=166.7  +MOVJ EC00115
SREFP 3 C00116 BC00116  +REFP EC00116
CALL JOB:SEARCH-R1-S13D
SET P032 P006
SFTON3D P032
SMOVL C00117 BC00117 V=166.7  +MOVJ EC00117
SMOVL C00118 BC00118 V=166.7  +MOVJ EC00118
SREFP 3 C00119 BC00119  +REFP EC00119
CALL JOB:SEARCH-R1-S13D
SET P032 P006
SFTON3D P032
SMOVL C00120 BC00120 V=166.7  +MOVJ EC00120
MOVL C00121 BC00121 V=800.0  +MOVJ EC00121 VJ=100.00
MOVL C00122 BC00122 V=1000.0  +MOVJ EC00122 VJ=100.00
'EndPath S4666
MOVJ C00123 BC00123 VJ=100.00  +MOVJ EC00123 VJ=100.00
'Path S3857
SFTOF3D
MOVJ C00124 BC00124 VJ=100.00  +MOVJ EC00124 VJ=100.00
MOVL C00125 BC00125 V=800.0  +MOVJ EC00125 VJ=100.00
SMOVL C00126 BC00126 V=166.7  +MOVJ EC00126
SREFP 3 C00127 BC00127  +REFP EC00127
CALL JOB:SEARCH-R1-S13D
SET P033 P006
SFTON3D P033
SMOVL C00128 BC00128 V=166.7  +MOVJ EC00128
SMOVL C00129 BC00129 V=166.7  +MOVJ EC00129
SREFP 3 C00130 BC00130  +REFP EC00130
CALL JOB:SEARCH-R1-S13D
SET P033 P006
SFTON3D P033
SMOVL C00131 BC00131 V=166.7  +MOVJ EC00131
SMOVL C00132 BC00132 V=166.7  +MOVJ EC00132
SREFP 3 C00133 BC00133  +REFP EC00133
CALL JOB:SEARCH-R1-S13D
SET P033 P006
SFTON3D P033
SMOVL C00134 BC00134 V=166.7  +MOVJ EC00134
MOVL C00135 BC00135 V=800.0  +MOVJ EC00135 VJ=100.00
MOVL C00136 BC00136 V=1000.0  +MOVJ EC00136 VJ=100.00
MOVL C00137 BC00137 V=1000.0  +MOVJ EC00137 VJ=100.00
'EndPath S3857
MOVJ C00138 BC00138 VJ=100.00  +MOVJ EC00138 VJ=100.00
'Path S4667
SFTOF3D
MOVJ C00139 BC00139 VJ=100.00  +MOVJ EC00139 VJ=100.00
MOVL C00140 BC00140 V=800.0  +MOVJ EC00140 VJ=100.00
SMOVL C00141 BC00141 V=166.7  +MOVJ EC00141
SREFP 3 C00142 BC00142  +REFP EC00142
CALL JOB:SEARCH-R1-S13D
SET P034 P006
SFTON3D P034
SMOVL C00143 BC00143 V=166.7  +MOVJ EC00143
SMOVL C00144 BC00144 V=166.7  +MOVJ EC00144
SREFP 3 C00145 BC00145  +REFP EC00145
CALL JOB:SEARCH-R1-S13D
SET P034 P006
SFTON3D P034
SMOVL C00146 BC00146 V=166.7  +MOVJ EC00146
SREFP 3 C00147 BC00147  +REFP EC00147
CALL JOB:SEARCH-R1-S13D
SET P034 P006
SFTON3D P034
SMOVL C00148 BC00148 V=166.7  +MOVJ EC00148
MOVL C00149 BC00149 V=800.0  +MOVJ EC00149 VJ=100.00
MOVL C00150 BC00150 V=1000.0  +MOVJ EC00150 VJ=100.00
MOVL C00151 BC00151 V=1000.0  +MOVJ EC00151 VJ=100.00
'EndPath S4667
MOVJ C00152 BC00152 VJ=100.00  +MOVJ EC00152 VJ=100.00
'Path S4668
SFTOF3D
MOVJ C00153 BC00153 VJ=100.00  +MOVJ EC00153 VJ=100.00
MOVL C00154 BC00154 V=800.0  +MOVJ EC00154 VJ=100.00
SMOVL C00155 BC00155 V=166.7  +MOVJ EC00155
SREFP 3 C00156 BC00156  +REFP EC00156
CALL JOB:SEARCH-R1-S13D
SET P035 P006
SFTON3D P035
SMOVL C00157 BC00157 V=166.7  +MOVJ EC00157
SMOVL C00158 BC00158 V=166.7  +MOVJ EC00158
SREFP 3 C00159 BC00159  +REFP EC00159
CALL JOB:SEARCH-R1-S13D
SET P035 P006
SFTON3D P035
SMOVL C00160 BC00160 V=166.7  +MOVJ EC00160
SMOVL C00161 BC00161 V=166.7  +MOVJ EC00161
SREFP 3 C00162 BC00162  +REFP EC00162
CALL JOB:SEARCH-R1-S13D
SET P035 P006
SFTON3D P035
SMOVL C00163 BC00163 V=166.7  +MOVJ EC00163
MOVL C00164 BC00164 V=800.0  +MOVJ EC00164 VJ=100.00
MOVL C00165 BC00165 V=1000.0  +MOVJ EC00165 VJ=100.00
'EndPath S4668
MOVJ C00166 BC00166 VJ=100.00  +MOVJ EC00166 VJ=100.00
'Path S4669
SFTOF3D
MOVJ C00167 BC00167 VJ=100.00  +MOVJ EC00167 VJ=100.00
MOVL C00168 BC00168 V=800.0  +MOVJ EC00168 VJ=100.00
SMOVL C00169 BC00169 V=166.7  +MOVJ EC00169
SREFP 3 C00170 BC00170  +REFP EC00170
CALL JOB:SEARCH-R1-S13D
SET P036 P006
SFTON3D P036
SMOVL C00171 BC00171 V=166.7  +MOVJ EC00171
SMOVL C00172 BC00172 V=166.7  +MOVJ EC00172
SREFP 3 C00173 BC00173  +REFP EC00173
CALL JOB:SEARCH-R1-S13D
SET P036 P006
SFTON3D P036
SMOVL C00174 BC00174 V=166.7  +MOVJ EC00174
SMOVL C00175 BC00175 V=166.7  +MOVJ EC00175
SREFP 3 C00176 BC00176  +REFP EC00176
CALL JOB:SEARCH-R1-S13D
SET P036 P006
SFTON3D P036
SMOVL C00177 BC00177 V=166.7  +MOVJ EC00177
MOVL C00178 BC00178 V=800.0  +MOVJ EC00178 VJ=100.00
MOVL C00179 BC00179 V=1000.0  +MOVJ EC00179 VJ=100.00
'EndPath S4669
MOVJ C00180 BC00180 VJ=100.00  +MOVJ EC00180 VJ=100.00
'Path S3859
SFTOF3D
MOVJ C00181 BC00181 VJ=100.00  +MOVJ EC00181 VJ=100.00
MOVL C00182 BC00182 V=800.0  +MOVJ EC00182 VJ=100.00
SMOVL C00183 BC00183 V=166.7  +MOVJ EC00183
SREFP 3 C00184 BC00184  +REFP EC00184
CALL JOB:SEARCH-R1-S13D
SET P037 P006
SFTON3D P037
SMOVL C00185 BC00185 V=166.7  +MOVJ EC00185
SMOVL C00186 BC00186 V=166.7  +MOVJ EC00186
SREFP 3 C00187 BC00187  +REFP EC00187
CALL JOB:SEARCH-R1-S13D
SET P037 P006
SFTON3D P037
SMOVL C00188 BC00188 V=166.7  +MOVJ EC00188
SMOVL C00189 BC00189 V=166.7  +MOVJ EC00189
SREFP 3 C00190 BC00190  +REFP EC00190
CALL JOB:SEARCH-R1-S13D
SET P037 P006
SFTON3D P037
SMOVL C00191 BC00191 V=166.7  +MOVJ EC00191
MOVL C00192 BC00192 V=800.0  +MOVJ EC00192 VJ=100.00
MOVL C00193 BC00193 V=1000.0  +MOVJ EC00193 VJ=100.00
'EndPath S3859
MOVJ C00194 BC00194 VJ=100.00  +MOVJ EC00194 VJ=100.00
'Path S4670
SFTOF3D
MOVJ C00195 BC00195 VJ=100.00  +MOVJ EC00195 VJ=100.00
MOVL C00196 BC00196 V=800.0  +MOVJ EC00196 VJ=100.00
SMOVL C00197 BC00197 V=166.7  +MOVJ EC00197
SREFP 3 C00198 BC00198  +REFP EC00198
CALL JOB:SEARCH-R1-S13D
SET P038 P006
SFTON3D P038
SMOVL C00199 BC00199 V=166.7  +MOVJ EC00199
SMOVL C00200 BC00200 V=166.7  +MOVJ EC00200
SREFP 3 C00201 BC00201  +REFP EC00201
CALL JOB:SEARCH-R1-S13D
SET P038 P006
SFTON3D P038
SMOVL C00202 BC00202 V=166.7  +MOVJ EC00202
SMOVL C00203 BC00203 V=166.7  +MOVJ EC00203
SREFP 3 C00204 BC00204  +REFP EC00204
CALL JOB:SEARCH-R1-S13D
SET P038 P006
SFTON3D P038
SMOVL C00205 BC00205 V=166.7  +MOVJ EC00205
MOVL C00206 BC00206 V=800.0  +MOVJ EC00206 VJ=100.00
MOVL C00207 BC00207 V=1000.0  +MOVJ EC00207 VJ=100.00
'EndPath S4670
MOVJ C00208 BC00208 VJ=100.00  +MOVJ EC00208 VJ=100.00
'Path S3860
SFTOF3D
MOVJ C00209 BC00209 VJ=100.00  +MOVJ EC00209 VJ=100.00
MOVL C00210 BC00210 V=800.0  +MOVJ EC00210 VJ=100.00
SMOVL C00211 BC00211 V=166.7  +MOVJ EC00211
SREFP 3 C00212 BC00212  +REFP EC00212
CALL JOB:SEARCH-R1-S13D
SET P039 P006
SFTON3D P039
SMOVL C00213 BC00213 V=166.7  +MOVJ EC00213
SMOVL C00214 BC00214 V=166.7  +MOVJ EC00214
SREFP 3 C00215 BC00215  +REFP EC00215
CALL JOB:SEARCH-R1-S13D
SET P039 P006
SFTON3D P039
SMOVL C00216 BC00216 V=166.7  +MOVJ EC00216
SMOVL C00217 BC00217 V=166.7  +MOVJ EC00217
SREFP 3 C00218 BC00218  +REFP EC00218
CALL JOB:SEARCH-R1-S13D
SET P039 P006
SFTON3D P039
SMOVL C00219 BC00219 V=166.7  +MOVJ EC00219
MOVL C00220 BC00220 V=800.0  +MOVJ EC00220 VJ=100.00
MOVL C00221 BC00221 V=1000.0  +MOVJ EC00221 VJ=100.00
'EndPath S3860
'Path S4671
SFTOF3D
MOVJ C00222 BC00222 VJ=100.00  +MOVJ EC00222 VJ=100.00
MOVL C00223 BC00223 V=800.0  +MOVJ EC00223 VJ=100.00
SMOVL C00224 BC00224 V=166.7  +MOVJ EC00224
SREFP 3 C00225 BC00225  +REFP EC00225
CALL JOB:SEARCH-R1-S13D
SET P040 P006
SFTON3D P040
SMOVL C00226 BC00226 V=166.7  +MOVJ EC00226
SMOVL C00227 BC00227 V=166.7  +MOVJ EC00227
SREFP 3 C00228 BC00228  +REFP EC00228
CALL JOB:SEARCH-R1-S13D
SET P040 P006
SFTON3D P040
SMOVL C00229 BC00229 V=166.7  +MOVJ EC00229
MOVL C00230 BC00230 V=800.0  +MOVJ EC00230 VJ=100.00
MOVL C00231 BC00231 V=1000.0  +MOVJ EC00231 VJ=100.00
'EndPath S4671
'Path W3861
SFTOF3D
SFTON3D P039
MOVJ C00232 BC00232 VJ=100.00  +MOVJ EC00232 VJ=100.00
SMOVL C00233 BC00233 V=800.0  +MOVJ EC00233
SMOVL C00234 BC00234 V=166.7 PL=0  +MOVJ EC00234
MACRO1 MJ#(0) ARGF9
ARCON
SMOVL C00235 BC00235 V=7.5  +MOVJ EC00235
SFTON3D P040
SMOVL C00236 BC00236 V=7.5  +MOVJ EC00236
SMOVL C00237 BC00237 V=7.5  +MOVJ EC00237
ARCOF
SMOVL C00238 BC00238 V=800.0  +MOVJ EC00238
SMOVL C00239 BC00239 V=1000.0  +MOVJ EC00239
SFTOF3D
'EndPath W3861
MOVJ C00240 BC00240 VJ=100.00  +MOVJ EC00240 VJ=100.00
'Path W3862
SFTOF3D
SFTON3D P037
MOVJ C00241 BC00241 VJ=100.00  +MOVJ EC00241 VJ=100.00
MOVJ C00242 BC00242 VJ=100.00  +MOVJ EC00242 VJ=100.00
SMOVL C00243 BC00243 V=800.0  +MOVJ EC00243
SMOVL C00244 BC00244 V=166.7 PL=0  +MOVJ EC00244
MACRO1 MJ#(0) ARGF14
ARCON
SMOVL C00245 BC00245 V=10.0  +MOVJ EC00245
SMOVL C00246 BC00246 V=10.0  +MOVJ EC00246
SFTON3D P038
SMOVL C00247 BC00247 V=10.0  +MOVJ EC00247
SMOVL C00248 BC00248 V=10.0  +MOVJ EC00248
ARCOF
SMOVL C00249 BC00249 V=800.0  +MOVJ EC00249
SMOVL C00250 BC00250 V=1000.0  +MOVJ EC00250
SFTOF3D
'EndPath W3862
MOVJ C00251 BC00251 VJ=100.00  +MOVJ EC00251 VJ=100.00
MOVJ C00252 BC00252 VJ=100.00  +MOVJ EC00252 VJ=100.00
'Path W3863
SFTOF3D
SFTON3D P035
MOVJ C00253 BC00253 VJ=100.00  +MOVJ EC00253 VJ=100.00
MOVJ C00254 BC00254 VJ=100.00  +MOVJ EC00254 VJ=100.00
SMOVL C00255 BC00255 V=800.0  +MOVJ EC00255
SMOVL C00256 BC00256 V=166.7 PL=0  +MOVJ EC00256
ARCON
SMOVL C00257 BC00257 V=9.2  +MOVJ EC00257
SFTON3D P036
SMOVL C00258 BC00258 V=9.2  +MOVJ EC00258
SMOVL C00259 BC00259 V=9.2  +MOVJ EC00259
ARCOF
SMOVL C00260 BC00260 V=800.0  +MOVJ EC00260
SMOVL C00261 BC00261 V=1000.0  +MOVJ EC00261
SMOVL C00262 BC00262 V=1000.0  +MOVJ EC00262
SFTOF3D
'EndPath W3863
MOVJ C00263 BC00263 VJ=100.00  +MOVJ EC00263 VJ=100.00
MOVJ C00264 BC00264 VJ=100.00  +MOVJ EC00264 VJ=100.00
'Path W3864
SFTOF3D
SFTON3D P033
MOVJ C00265 BC00265 VJ=100.00  +MOVJ EC00265 VJ=100.00
SMOVL C00266 BC00266 V=800.0  +MOVJ EC00266
SMOVL C00267 BC00267 V=166.7 PL=0  +MOVJ EC00267
ARCON
SMOVL C00268 BC00268 V=10.0  +MOVJ EC00268
SFTON3D P034
SMOVL C00269 BC00269 V=10.0  +MOVJ EC00269
SMOVL C00270 BC00270 V=10.0  +MOVJ EC00270
ARCOF
SMOVL C00271 BC00271 V=800.0  +MOVJ EC00271
SMOVL C00272 BC00272 V=1000.0  +MOVJ EC00272
SMOVL C00273 BC00273 V=1000.0  +MOVJ EC00273
SFTOF3D
'EndPath W3864
MOVJ C00274 BC00274 VJ=100.00  +MOVJ EC00274 VJ=100.00
'Path W3865
SFTOF3D
SFTON3D P032
MOVJ C00275 BC00275 VJ=100.00  +MOVJ EC00275 VJ=100.00
MOVJ C00276 BC00276 VJ=100.00  +MOVJ EC00276 VJ=100.00
SMOVL C00277 BC00277 V=800.0  +MOVJ EC00277
SMOVL C00278 BC00278 V=166.7 PL=0  +MOVJ EC00278
ARCON
SMOVL C00279 BC00279 V=9.2  +MOVJ EC00279
SFTON3D P031
SMOVL C00280 BC00280 V=9.2  +MOVJ EC00280
SMOVL C00281 BC00281 V=9.2  +MOVJ EC00281
ARCOF
SMOVL C00282 BC00282 V=800.0  +MOVJ EC00282
SMOVL C00283 BC00283 V=1000.0  +MOVJ EC00283
SFTOF3D
'EndPath W3865
MOVJ C00284 BC00284 VJ=100.00  +MOVJ EC00284 VJ=100.00
'Down
MOVJ C00285 BC00285 VJ=100.00  +MOVJ EC00285 VJ=100.00
MOVJ C00286 BC00286 VJ=100.00  +MOVJ EC00286 VJ=100.00
'Path W3867
SFTOF3D
SFTON3D P026
MOVJ C00287 BC00287 VJ=100.00  +MOVJ EC00287 VJ=100.00
SMOVL C00288 BC00288 V=800.0  +MOVJ EC00288
SMOVL C00289 BC00289 V=150.0 PL=0  +MOVJ EC00289
MACRO1 MJ#(0) ARGF22
ARCON
SMOVC C00290 BC00290 V=9.5  +MOVJ EC00290
SMOVC C00291 BC00291 V=9.5  +MOVJ EC00291
SFTON3D P025
SMOVC C00292 BC00292 V=9.5  +MOVJ EC00292
SMOVL C00293 BC00293 V=9.5  +MOVJ EC00293
ARCOF
SMOVL C00294 BC00294 V=800.0  +MOVJ EC00294
SMOVL C00295 BC00295 V=1000.0  +MOVJ EC00295
SFTOF3D
'EndPath W3867
MOVJ C00296 BC00296 VJ=100.00  +MOVJ EC00296 VJ=100.00
MOVJ C00297 BC00297 VJ=100.00  +MOVJ EC00297 VJ=100.00
MOVJ C00298 BC00298 VJ=100.00  +MOVJ EC00298 VJ=100.00
'Path W3868
SFTOF3D
SFTON3D P022
MOVJ C00299 BC00299 VJ=100.00  +MOVJ EC00299 VJ=100.00
MOVJ C00300 BC00300 VJ=100.00  +MOVJ EC00300 VJ=100.00
SMOVL C00301 BC00301 V=800.0  +MOVJ EC00301
SMOVL C00302 BC00302 V=166.7 PL=0  +MOVJ EC00302
MACRO1 MJ#(0) ARGF9
ARCON
SMOVL C00303 BC00303 V=10.0  +MOVJ EC00303
SMOVL C00304 BC00304 V=10.0  +MOVJ EC00304
SMOVL C00305 BC00305 V=10.0  +MOVJ EC00305
SMOVL C00306 BC00306 V=10.0  +MOVJ EC00306
SMOVL C00307 BC00307 V=10.0  +MOVJ EC00307
SMOVL C00308 BC00308 V=10.0  +MOVJ EC00308
SMOVL C00309 BC00309 V=10.0  +MOVJ EC00309
SMOVL C00310 BC00310 V=10.0  +MOVJ EC00310
SMOVL C00311 BC00311 V=10.0  +MOVJ EC00311
ARCOF
SMOVL C00312 BC00312 V=800.0  +MOVJ EC00312
SMOVL C00313 BC00313 V=1000.0  +MOVJ EC00313
SFTOF3D
'EndPath W3868
MOVJ C00314 BC00314 VJ=100.00  +MOVJ EC00314 VJ=100.00
SFTOF3D
'EndPath W3869
MOVJ C00315 BC00315 VJ=100.00  +MOVJ EC00315 VJ=100.00
'Path W3896
SFTOF3D
SFTON3D P020
MOVJ C00316 BC00316 VJ=100.00  +MOVJ EC00316 VJ=100.00
SMOVL C00317 BC00317 V=800.0  +MOVJ EC00317
SMOVL C00318 BC00318 V=150.0 PL=0  +MOVJ EC00318
ARCON
SMOVL C00319 BC00319 V=10.0  +MOVJ EC00319
SMOVL C00320 BC00320 V=10.0  +MOVJ EC00320
ARCOF
SMOVL C00321 BC00321 V=800.0  +MOVJ EC00321
SFTOF3D
'EndPath W3896
MOVJ C00322 BC00322 VJ=100.00  +MOVJ EC00322 VJ=100.00
MOVJ C00323 BC00323 VJ=100.00  +MOVJ EC00323 VJ=100.00
MOVJ C00324 BC00324 VJ=100.00  +MOVJ EC00324 VJ=100.00
'Path W3866
SFTOF3D
SFTON3D P023
MOVJ C00325 BC00325 VJ=100.00  +MOVJ EC00325 VJ=100.00
SMOVL C00326 BC00326 V=800.0  +MOVJ EC00326
SMOVC C00327 BC00327 V=150.0 PL=0  +MOVJ EC00327
MACRO1 MJ#(0) ARGF22
ARCON
SWVON WEV#(108)
SMOVC C00328 BC00328 V=9.5  +MOVJ EC00328
SMOVC C00329 BC00329 V=9.5  +MOVJ EC00329
SFTON3D P024
SMOVC C00330 BC00330 V=9.5  +MOVJ EC00330
SMOVC C00331 BC00331 V=9.5  +MOVJ EC00331
ARCOF
SWVOF
SMOVL C00332 BC00332 V=800.0  +MOVJ EC00332
SMOVL C00333 BC00333 V=1000.0  +MOVJ EC00333
SFTOF3D
'EndPath W3866
MOVJ C00334 BC00334 VJ=100.00  +MOVJ EC00334 VJ=100.00
'jakie searche do takicj spoin?
'kamera
MOVJ C00335 BC00335 VJ=100.00  +MOVJ EC00335 VJ=100.00
SFTOF3D
'EndPath W3891
'jakie searche do takicj spoin?
'68,69
MOVJ C00336 BC00336 VJ=20.00  +MOVJ EC00336 VJ=20.00
MOVJ C00337 BC00337 VJ=100.00  +MOVJ EC00337 VJ=100.00
'Path W4660
SFTOF3D
COMM SFTON3D P041
COMM MOVJ C00338 BC00338 VJ=100.00  +MOVJ EC00338 VJ=100.00
COMM SMOVL C00339 BC00339 V=800.0  +MOVJ EC00339
COMM SMOVL C00340 BC00340 V=150.0 PL=0  +MOVJ EC00340
COMM MACRO1 MJ#(0) ARGF9
COMM ARCON
COMM SMOVL C00341 BC00341 V=11.7  +MOVJ EC00341
COMM ARCOF
COMM SMOVL C00342 BC00342 V=800.0  +MOVJ EC00342
COMM SMOVL C00343 BC00343 V=1000.0  +MOVJ EC00343
COMM SFTOF3D
COMM 'EndPath W4660
COMM 'Path W4662
COMM SFTOF3D
COMM SFTON3D P042
COMM MOVJ C00344 BC00344 VJ=100.00  +MOVJ EC00344 VJ=100.00
COMM SMOVL C00345 BC00345 V=800.0  +MOVJ EC00345
COMM SMOVL C00346 BC00346 V=150.0 PL=0  +MOVJ EC00346
COMM ARCON
COMM SMOVL C00347 BC00347 V=11.7  +MOVJ EC00347
COMM ARCOF
COMM SMOVL C00348 BC00348 V=800.0  +MOVJ EC00348
SMOVL C00349 BC00349 V=1000.0  +MOVJ EC00349
SMOVL C00350 BC00350 V=1000.0  +MOVJ EC00350
SFTOF3D
'EndPath W4662
'Path W3893
SFTOF3D
MOVJ C00351 BC00351 VJ=100.00  +MOVJ EC00351 VJ=100.00
MOVJ C00352 BC00352 VJ=100.00  +MOVJ EC00352 VJ=100.00
MOVL C00353 BC00353 V=800.0  +MOVJ EC00353 VJ=100.00
SMOVL C00354 BC00354 V=166.7 PL=0  +MOVJ EC00354
MACRO1 MJ#(0) ARGF20
ARCON
SMOVL C00355 BC00355 V=6.7  +MOVJ EC00355
SMOVL C00356 BC00356 V=6.7  +MOVJ EC00356
SMOVL C00357 BC00357 V=6.7  +MOVJ EC00357
ARCOF
SWVOF
SFTOF3D
MOVL C00358 BC00358 V=800.0  +MOVJ EC00358 VJ=100.00
MOVL C00359 BC00359 V=1000.0  +MOVJ EC00359 VJ=100.00
MOVL C00360 BC00360 V=1000.0  +MOVJ EC00360 VJ=100.00
'EndPath W3893
'68,69
MOVJ C00361 BC00361 VJ=100.00  +MOVJ EC00361 VJ=100.00
MOVJ C00362 BC00362 VJ=100.00  +MOVJ EC00362 VJ=100.00
MOVJ C00363 BC00363 VJ=100.00  +MOVJ EC00363 VJ=100.00
'
END
